// TIA Portal V16 export
// export: Created 2022-02-28T20:45:42.6040765Z, ExportSetting WithDefaults, DisplayName Totally Integrated Automation Portal, DisplayVersion V16, DisplayName TIA Portal Version Control Interface, DisplayVersion V16, DisplayName TIA Portal Openness, DisplayVersion V16, DisplayName STEP 7 Professional, DisplayVersion V16, DisplayName STEP 7 Safety, DisplayVersion V16, DisplayName WinCC Advanced, DisplayVersion V16
ORGANIZATION_BLOCK "Main"   // OB1, LAD, ProgramCycle
TITLE = "Main Program Sweep (Cycle)"
{ S7_Optimized_Access := 'TRUE' }
VERSION : 0.1
// stored: AutoNumber true, IsIECCheckEnabled false, SetENOAutomatically false
   VAR_INPUT
      Initial_Call : Bool;   // Initial call of this OB
      Remanence : Bool;   // =True, if remanent data are available
   END_VAR
   VAR_TEMP   // added for the SCL form of the ladder/FBD networks
      _w1 : Bool;
      _w2 : Bool;
   END_VAR
BEGIN

REGION Network 1
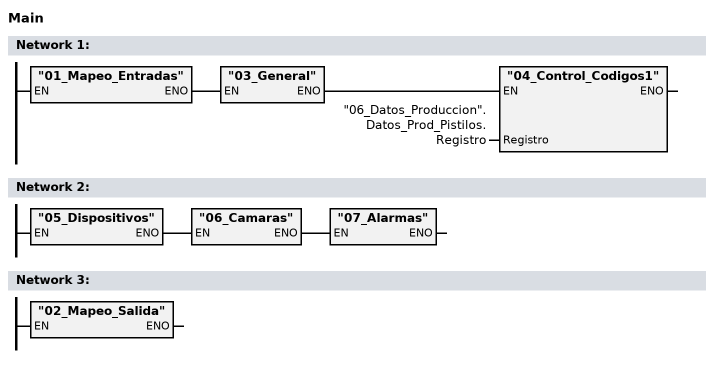
   RUNG wire#powerrail
      "01_Mapeo_Entradas"()
      "03_General"()
      "04_Control_Codigos1"(Registro := "06_Datos_Produccion".Datos_Prod_Pistilos.Registro)
   END_RUNG
   // the same network as SCL:
   "01_Mapeo_Entradas"(ENO => #_w1);
   "03_General"(EN := #_w1, ENO => #_w2);
   IF #_w2 THEN
       "04_Control_Codigos1"(Registro := "06_Datos_Produccion".Datos_Prod_Pistilos.Registro);
   END_IF;
END_REGION

REGION Network 2
   RUNG wire#powerrail
      "05_Dispositivos"()
      "06_Camaras"()
      "07_Alarmas"()
   END_RUNG
   // the same network as SCL:
   "05_Dispositivos"(ENO => #_w1);
   "06_Camaras"(EN := #_w1, ENO => #_w2);
   IF #_w2 THEN "07_Alarmas"(); END_IF;
END_REGION

REGION Network 3
   RUNG wire#powerrail
      "02_Mapeo_Salida"()
   END_RUNG
   // the same network as SCL:
   "02_Mapeo_Salida"();
END_REGION
END_ORGANIZATION_BLOCK
